// TIA Portal V17 export
// export: Created 2021-09-08T12:46:16.1780561Z, ExportSetting WithDefaults, DisplayName Totally Integrated Automation Portal, DisplayVersion V17, DisplayName TIA Portal Openness, DisplayVersion V17, DisplayName TIA Portal Version Control Interface, DisplayVersion V17, DisplayName STEP 7 Professional, DisplayVersion V17, DisplayName STEP 7 Safety, DisplayVersion V17, DisplayName WinCC Advanced, DisplayVersion V17
FUNCTION "Multiply" : Void   // FC0, LAD
TITLE = Multiply
{ S7_Optimized_Access := 'TRUE' }
VERSION : 1.1
// Some Comment
// stored: AutoNumber true, IsIECCheckEnabled false, SetENOAutomatically false, StructureModified 2022-04-29T09:29:23, UDAEnableTagReadback false
   VAR_INPUT
      In1 : Real;
      In2 : Real;
   END_VAR
   VAR_OUTPUT
      Out : Real;
   END_VAR
BEGIN

REGION Network 1: Multiply
   // Some Comment
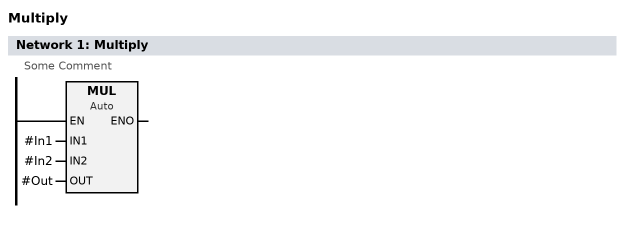
   RUNG wire#powerrail
      { S7_GenerateENO := "TRUE" } Mul(in1 := #In1, in2 := #In2, out := #Out)
   END_RUNG
   // the same network as SCL:
   <??.?> := #In1 * #In2 * #Out;
END_REGION
END_FUNCTION
